// TIA Portal V15.1 export
// export: Created 2020-06-12T07:35:42.1630859Z, ExportSetting None, DisplayName Totally Integrated Automation Portal, DisplayVersion V15.1, DisplayName TIA Portal Openness, DisplayVersion V15.1, DisplayName STEP 7 Professional, DisplayVersion V15.1, DisplayName STEP 7 Safety, DisplayVersion V15.1, DisplayName WinCC Advanced, DisplayVersion V15.1
FUNCTION "ES1_field" : Void   // FC78, FBD
TITLE = Field devices: monitoring and control
{ S7_Optimized_Access := 'TRUE' }
// * I/O part
// * Control part
// stored: SetENOAutomatically False
BEGIN

REGION Network 1: Safety states monitoring
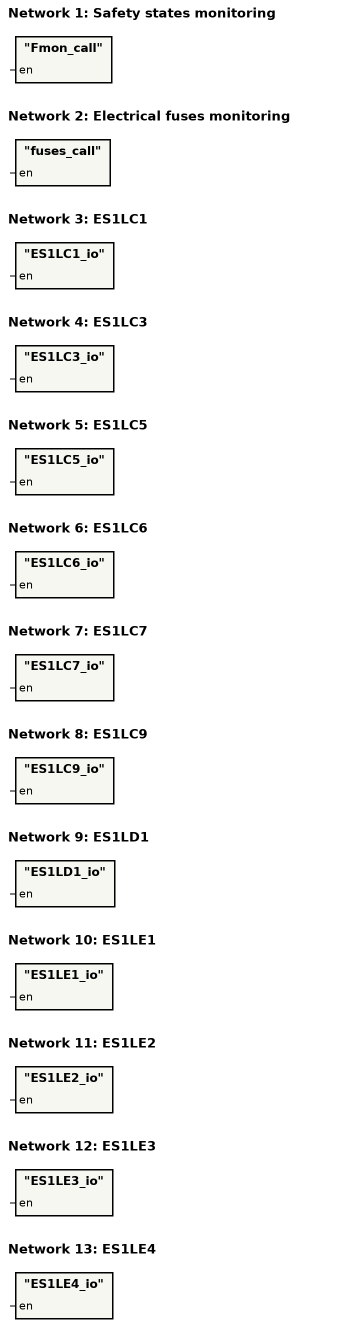
   "Fmon_call"();
END_REGION

REGION Network 2: Electrical fuses monitoring
   "fuses_call"();
END_REGION

REGION Network 3: ES1LC1
   "ES1LC1_io"();
END_REGION

REGION Network 4: ES1LC3
   "ES1LC3_io"();
END_REGION

REGION Network 5: ES1LC5
   "ES1LC5_io"();
END_REGION

REGION Network 6: ES1LC6
   "ES1LC6_io"();
END_REGION

REGION Network 7: ES1LC7
   "ES1LC7_io"();
END_REGION

REGION Network 8: ES1LC9
   "ES1LC9_io"();
END_REGION

REGION Network 9: ES1LD1
   "ES1LD1_io"();
END_REGION

REGION Network 10: ES1LE1
   "ES1LE1_io"();
END_REGION

REGION Network 11: ES1LE2
   "ES1LE2_io"();
END_REGION

REGION Network 12: ES1LE3
   "ES1LE3_io"();
END_REGION

REGION Network 13: ES1LE4
   "ES1LE4_io"();
END_REGION

REGION Network 14: ES1LG1
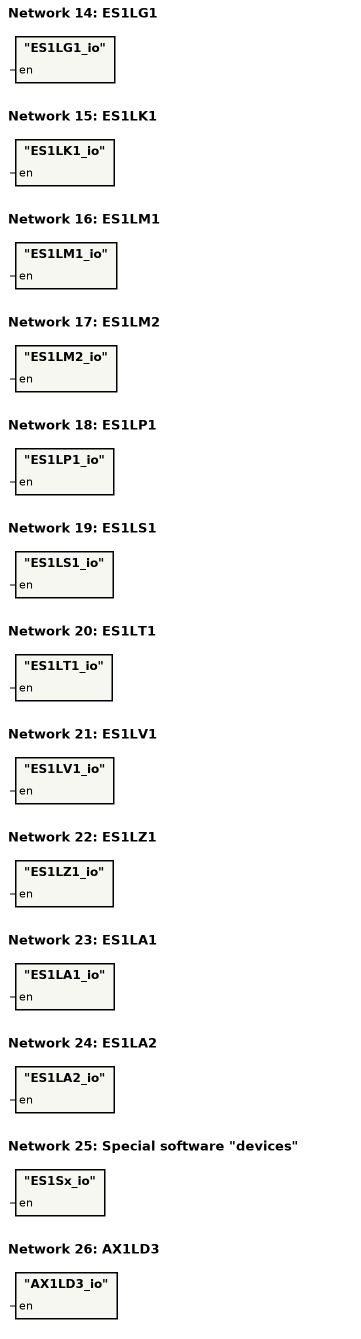
   "ES1LG1_io"();
END_REGION

REGION Network 15: ES1LK1
   "ES1LK1_io"();
END_REGION

REGION Network 16: ES1LM1
   "ES1LM1_io"();
END_REGION

REGION Network 17: ES1LM2
   "ES1LM2_io"();
END_REGION

REGION Network 18: ES1LP1
   "ES1LP1_io"();
END_REGION

REGION Network 19: ES1LS1
   "ES1LS1_io"();
END_REGION

REGION Network 20: ES1LT1
   "ES1LT1_io"();
END_REGION

REGION Network 21: ES1LV1
   "ES1LV1_io"();
END_REGION

REGION Network 22: ES1LZ1
   "ES1LZ1_io"();
END_REGION

REGION Network 23: ES1LA1
   "ES1LA1_io"();
END_REGION

REGION Network 24: ES1LA2
   "ES1LA2_io"();
END_REGION

REGION Network 25: Special software "devices"
   "ES1Sx_io"();
END_REGION

REGION Network 26: AX1LD3
   "AX1LD3_io"();
END_REGION
END_FUNCTION
